// TIA Portal project "Birden Fazla Konvenyör Bandı Çalıştırma Ve Check Box Kullanım Mantığı_V15.1" (V15.1)
// Vorlageprojekt für das Buch mit Zielsystem S7-1200

(* hardware
DEVICE "S7-1200-Station_1"  S7-1200 Station
   slot 0: "Baugruppenträger_0"  Rack  V1.0
   slot 1: "PLC_1"  CPU 1211C DC/DC/DC  6ES7 211-1AE40-0XB0  V4.1
DEVICE "PC station"  SIMATIC PC station
   slot 0: "PC station"  Rail  SIMATIC PC-Station  V1.0
      slot 125: "Stationmanager"  Station_Manager  V6.0.4
   slot 1: "IE general_1"  IE General  IE_CP  V8.2.0
   slot 2: "HMI_RT_1"  WinCC RT Advanced  6AV2 104-0xxxx-xxxx  15.1.0.0
      slot 33792: "Host interface"  Host interface
*)

// ===== PLC "PLC_1"  CPU 1211C DC/DC/DC =====

VAR_GLOBAL   // PLC tag table "Standard-Variablentabelle"
   "start_stop" AT %I0.0 : Bool;
   "sistem_devrede" AT %M5.0 : Bool;
   "konv_1" AT %Q0.0 : Bool;
   "konv_2" AT %Q0.1 : Bool;
   "konv_3" AT %Q0.2 : Bool;
   "konv_4" AT %Q0.3 : Bool;
   "ikaz_lambasi_1" AT %Q0.4 : Bool;
   "ikaz_lambasi_2" AT %Q0.5 : Bool;
   "ikaz_lambasi_3" AT %Q0.6 : Bool;
   "start_up_mem" AT %M6.0 : Bool;
   "back" AT %M6.1 : Bool;
END_VAR

VAR_GLOBAL   // PLC tag table "hmi_tags"
   "hmi_start_stop" AT %M5.1 : Bool;
END_VAR

// folder: System blocks/Program resources

DATA_BLOCK "baslangıc_konumu"   // DB1
{ S7_Optimized_Access := 'TRUE' }
AUTHOR : Simatic
FAMILY : IEC
NAME : IEC_TMR
VERSION : 1.0
// stored: InstanceOfName IEC_TIMER
"IEC_TIMER"
BEGIN
END_DATA_BLOCK

DATA_BLOCK "sistem_calısma_suresi"   // DB2
{ S7_Optimized_Access := 'TRUE' }
AUTHOR : Simatic
FAMILY : IEC
NAME : IEC_TMR
VERSION : 1.0
// stored: InstanceOfName IEC_TIMER
"IEC_TIMER"
BEGIN
END_DATA_BLOCK

// folder: (top level)

FUNCTION "MHJ-PLC-Lab-Function-S71200" : Void   // FC9000, SCL
{ S7_Optimized_Access := 'TRUE' }
VERSION : 0.1
   VAR_TEMP
      rdTimeReturn : Int;
      outputTime : DTL;
      SyncVal : Byte;
      forVal : Int;
      forVal_2 : Int;
      Value : Byte;
   END_VAR
   VAR CONSTANT
      CompVal : Byte := 16#34;
      Value_01 : Byte := 16#11;
      Value_01_DW : DWord := 16#A165_D992;
      Value_02_DW : DWord := 16#58BE_4401;
   END_VAR
BEGIN

   #Value:=PEEK(area := 16#82,
        dbNumber := 0,
        byteOffset := 511);
   #Value := #Value + 1;

   POKE(area := 16#82,
        dbNumber := 0,
        byteOffset := 511,
        value := #Value);

   POKE(area:=16#81,
        dbNumber:=0,
        byteOffset:=1016,
        value:=#Value_01_DW);
   POKE(area := 16#81,
        dbNumber := 0,
        byteOffset := 1020,
        value := #Value_02_DW);

   POKE(area := 16#81,
        dbNumber := 0,
        byteOffset := 511,
        value := B#16#00);

   FOR #forVal := 0 TO 120 DO
       FOR #forVal_2:=0 TO 10 DO
           #rdTimeReturn:=RD_SYS_T(#outputTime);
           #rdTimeReturn := WR_SYS_T(#outputTime);
           #rdTimeReturn := RD_SYS_T(#outputTime);
           #rdTimeReturn := WR_SYS_T(#outputTime);
       END_FOR;
       #SyncVal:= PEEK(area := 16#81,
                      dbNumber := 0,
                      byteOffset := 511);
       IF #SyncVal = #CompVal THEN
          GOTO M_1;
       END_IF;
   END_FOR;
   RETURN;

   M_1:
   POKE(area := 16#81,
        dbNumber := 0,
        byteOffset := 511,
        value := B#16#0);
END_FUNCTION

ORGANIZATION_BLOCK "Main"   // OB1, LAD, ProgramCycle
TITLE = "Main Program Sweep (Cycle)"
{ S7_Optimized_Access := 'TRUE' }
VERSION : 0.1
   VAR_INPUT
      Initial_Call : Bool;   // Initial call of this OB
      Remanence : Bool;   // =True, if remanent data are available
   END_VAR
BEGIN

REGION Network 1: Konnektierungsbaustein für PLC-Lab
   // Im Netzwerk 1 wird der Konnektierungsbaustein für PLC-Lab aufgerufen.
   // Dieser Aufruf darf nicht entfernt werden!
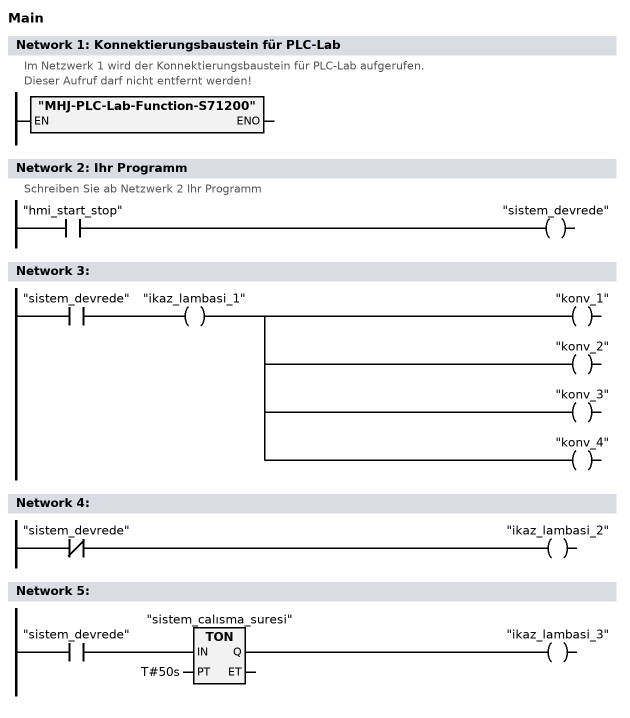
   RUNG wire#powerrail
      "MHJ-PLC-Lab-Function-S71200"()
   END_RUNG
   // the same network as SCL:
   "MHJ-PLC-Lab-Function-S71200"();
END_REGION

REGION Network 2: Ihr Programm
   // Schreiben Sie ab Netzwerk 2 Ihr Programm
   RUNG wire#powerrail
      Contact( "hmi_start_stop" )
      Coil( "sistem_devrede" )
   END_RUNG
   // the same network as SCL:
   "sistem_devrede" := "hmi_start_stop";
END_REGION

REGION Network 3
   RUNG wire#powerrail
      Contact( "sistem_devrede" )
      Coil( "ikaz_lambasi_1" )
      wire#w1
      Coil( "konv_1" )
   END_RUNG
   RUNG wire#w1
      Coil( "konv_2" )
   END_RUNG
   RUNG wire#w1
      Coil( "konv_3" )
   END_RUNG
   RUNG wire#w1
      Coil( "konv_4" )
   END_RUNG
   // the same network as SCL:
   "ikaz_lambasi_1" := "sistem_devrede";
   "konv_1" := "sistem_devrede";
   "konv_2" := "sistem_devrede";
   "konv_3" := "sistem_devrede";
   "konv_4" := "sistem_devrede";
END_REGION

REGION Network 4
   RUNG wire#powerrail
      I_Contact( "sistem_devrede" )
      Coil( "ikaz_lambasi_2" )
   END_RUNG
   // the same network as SCL:
   "ikaz_lambasi_2" := NOT "sistem_devrede";
END_REGION

REGION Network 5
   "sistem_calısma_suresi".TON(IN := "sistem_devrede", PT := T#50s);
   "ikaz_lambasi_3" := "sistem_calısma_suresi".Q;
END_REGION
END_ORGANIZATION_BLOCK

ORGANIZATION_BLOCK "Startup"   // OB100, LAD, Startup
TITLE = "Complete Restart"
{ S7_Optimized_Access := 'TRUE' }
VERSION : 0.1
   VAR_INPUT
      LostRetentive : Bool;   // True if retentive data are lost
      LostRTC : Bool;   // True if date and time are lost
   END_VAR
   VAR_TEMP
      start_up_mem : Bool;
   END_VAR
BEGIN

REGION Network 1
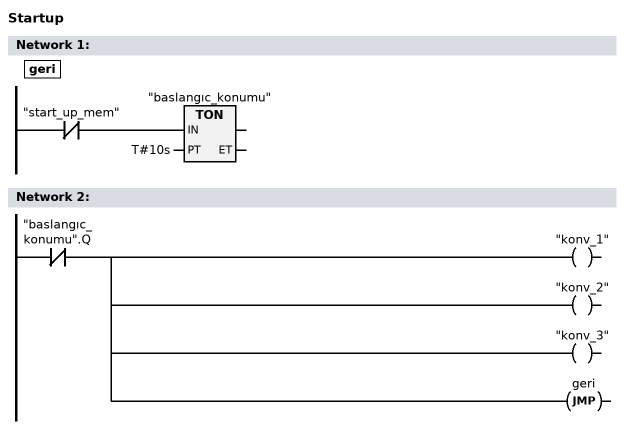
   geri:
   "baslangıc_konumu".TON(IN := NOT "start_up_mem", PT := T#10s);
END_REGION

REGION Network 2
   RUNG wire#powerrail
      I_Contact( "baslangıc_konumu".Q )
      wire#w1
      Coil( "konv_1" )
   END_RUNG
   RUNG wire#w1
      Coil( "konv_2" )
   END_RUNG
   RUNG wire#w1
      Coil( "konv_3" )
   END_RUNG
   RUNG wire#w1
      JumpCoil( geri )
   END_RUNG
   // the same network as SCL:
   "konv_1" := NOT "baslangıc_konumu".Q;
   "konv_2" := NOT "baslangıc_konumu".Q;
   "konv_3" := NOT "baslangıc_konumu".Q;
   IF NOT "baslangıc_konumu".Q THEN GOTO geri; END_IF;
END_REGION
END_ORGANIZATION_BLOCK

(* ===== HMI "HMI_RT_1" =====
system functions are stored by id; their names below are inferred from use
connection "HMI_Connection_1": ETHERNET, S7_1200_OMS

HMI tags "Default tag table"
   "hmi_start_stop" : Bool = PLC hmi_start_stop AT %M5.1, 1 s
   "sistem_devrede" : Bool = PLC sistem_devrede AT %M5.0, 1 s
   "ikaz_lambasi_3" : Bool = PLC ikaz_lambasi_3 AT %Q0.6, 1 s

screen "Screen_1" 1024x768
   GraphicView "Graphic view_1" at 288,192 size 300x300; Picture "Graphic_1"
   GraphicView "Graphic view_4" at 360,336 size 145x213; Picture "Graphic_4"
   Button "Button_1" at 64,96 size 176x48; TextOff 'START STOP'
      on Press: InvertBit("hmi_start_stop")
   Circle "Circle_1" at 376,376 size 32x32
      Appearance <- "sistem_devrede"
   Circle "Circle_2" at 416,376 size 32x32
      Appearance <- "sistem_devrede"
   Circle "Circle_3" at 456,376 size 32x32
      Appearance <- "ikaz_lambasi_3"
*)